Fanuc KAREL source: ka00105.KL

-- PROVISIONAL review KL for V770-1; original PC SHA256 38b0bd24827934f2d2388eb42b5be0585c0b6a66e13fa529f0cf09bfde0df22c
-- Incomplete behavior may be omitted. Consult companion uncertainty JSON. Do not deploy.
PROGRAM KA00105
%NOLOCKGROUP
-- UNRESOLVED_DECL SRC type=000013
-- UNRESOLVED_DECL DST type=000013
BEGIN
  -- UNRESOLVED_PC offsets 5-20; opcodes 2E,22,32,35
  -- UNRESOLVED_PC offsets 25-40; opcodes 49,4A
  -- UNRESOLVED_PC offsets 45-49; opcodes 7F
END KA00105
